// TIA Portal V17 export
// export: Created 2024-08-07T21:44:07.6081034Z, ExportSetting WithDefaults, DisplayName Totally Integrated Automation Portal, DisplayVersion V17 Update 7, DisplayName TIA Portal Openness, DisplayVersion V17 Update 7, DisplayName TIA Portal Version Control Interface, DisplayVersion V17, DisplayName SINAMICS Startdrive Advanced, DisplayVersion V17 SP2, DisplayName SINAMICS Startdrive G110M, G120, G120C, G120D, G120P, G115D, DisplayVersion V17 SP2, DisplayName SINAMICS Startdrive G130, G150, S120, S150, SINAMICS MV, S210, DisplayVersion V17 SP2, DisplayName STEP 7 Professional, DisplayVersion V17 Update 7, DisplayName STEP 7 Safety, DisplayVersion V17 Update 6, DisplayName WinCC Advanced / Unified PC, DisplayVersion V17 Update 7
DATA_BLOCK "PartsDataTransfer_DB"   // DB4
VERSION : 0.1
// stored: AutoNumber true, DBAccessibleFromOPCUA true, DBAccessibleFromWebserver true, InstanceOfName PartsDataTransfer, InstanceOfType FB
"PartsDataTransfer"
   // VAR
   //    gripperClose : R_TRIG;
   //    gripperOpen { S7_SetPoint := 'True'} : R_TRIG;
   //    gripperOpenPartial { S7_SetPoint := 'True'} : R_TRIG;
   // END_VAR
BEGIN
   gripperClose.CLK := FALSE;
   gripperClose.Q := FALSE;
   gripperClose.Stat_Bit := FALSE;
   gripperOpen.CLK := TRUE;
   gripperOpen.Q := FALSE;
   gripperOpen.Stat_Bit := TRUE;
   gripperOpenPartial.CLK := TRUE;
   gripperOpenPartial.Q := FALSE;
   gripperOpenPartial.Stat_Bit := TRUE;
END_DATA_BLOCK
